TEXTLIST TextList_MU_errorid
  0 = 'no_error'
  1 = 'not_connected'
  2 = 'invalid_state'
  3 = 'alarm_circulation_left'
  4 = 'alarm_circulation_right'
  5 = 'alarm_through_left'
  6 = 'alarm_through_right'
  7 = 'alarm_runtime_circulation_left'
  8 = 'alarm_runtime_circulation_right'
  9 = 'unknown_error'
  666 = 'emergency_error'
   = ''
END_TEXTLIST

(* stored: Version 1.1.0.1, ProductVersion 3.1.4024.11
   TextList TextList_MU_errorid: Id {47ca0037-1a21-4327-a432-6a08a9f274ae} *)
